KUKA KRL program: chk_w1_wechs_ok.src

&ACCESS RVO5
&REL 6
&COMMENT Check C1
DEF chk_w1_wechs_ok( )
;Diag_Appl(#on,5)

; VERIFICAÇÃO DE FERRAMENTA: C1

$TIMER[10] = 0
$TIMER_STOP[10] = FALSE

WAIT for ((not $in[161]) and (($in[169]) OR (NOT $in[169])) and ( $in[177]) and ( $in[185]) and ($in[219]))

;//---- End -------
;Diag_Appl(#Off,5)

$TIMER_STOP[10] = TRUE
$TIMER[10] = 0

END
